FUNCTION_BLOCK FB_Component_InductiveSensor_Test EXTENDS TcUnit.FB_TestSuite
VAR_INPUT
END_VAR
VAR_OUTPUT
END_VAR
VAR
END_VAR

AssertEquals(Expected := 1,
             Actual := 1,
             Message := 'The calculation is not correct');
TEST_FINISHED();

END_FUNCTION_BLOCK

(* stored: Version 1.1.0.1, ProductVersion 3.1.4024.15
   POU FB_Component_InductiveSensor_Test: Id {54a89a6a-35d4-4462-9810-666a8b15c961}, SpecialFunc None *)
